// TIA Portal V20 export
TYPE "typeCmHmiInterfaceBrakeTest"
// stored: Access Published, Namespace Unit1.Em2
   STRUCT
      jrOutPnPLeftAxisZ : "LER_typeBrakeTestEmInterface";
      jrOutPnPRightAxisZ : "LER_typeBrakeTestEmInterface";
   END_STRUCT;
END_TYPE
